// TIA Portal V17 export
// export: Created 2024-09-03T21:54:57.3136222Z, ExportSetting WithDefaults, DisplayName Totally Integrated Automation Portal, DisplayVersion V17 Update 7, DisplayName TIA Portal Openness, DisplayVersion V17 Update 7, DisplayName TIA Portal Version Control Interface, DisplayVersion V17, DisplayName SINAMICS Startdrive Advanced, DisplayVersion V17 SP2, DisplayName SINAMICS Startdrive G110M, G120, G120C, G120D, G120P, G115D, DisplayVersion V17 SP2, DisplayName SINAMICS Startdrive G130, G150, S120, S150, SINAMICS MV, S210, DisplayVersion V17 SP2, DisplayName STEP 7 Professional, DisplayVersion V17 Update 7, DisplayName STEP 7 Safety, DisplayVersion V17 Update 6, DisplayName WinCC Advanced / Unified PC, DisplayVersion V17 Update 7
DATA_BLOCK "AlarmsHandling_DB"   // DB16
VERSION : 0.1
// stored: AutoNumber true, DBAccessibleFromOPCUA true, DBAccessibleFromWebserver true, InstanceOfName AlarmsHandling, InstanceOfType FB
"AlarmsHandling"
   // VAR
   //    IEC_Timer_0_Instance_4 { S7_SetPoint := 'True'} : TON_TIME;
   //    IEC_Timer_0_Instance_5 { S7_SetPoint := 'True'} : TP_TIME;
   //    SetAlarmInstance { S7_SetPoint := 'True'} : Array[0..100] of "SetAlarm_PLC";
   //    AlarmPLCset { S7_SetPoint := 'True'} : Array[0..100] of Program_Alarm;
   // END_VAR
BEGIN
   IEC_Timer_0_Instance_4.PT := T#3S;
   IEC_Timer_0_Instance_4.IN := FALSE;
   IEC_Timer_0_Instance_5.PT := T#0MS;
   IEC_Timer_0_Instance_5.IN := FALSE;
   SetAlarmInstance[0..100].iAlarmCondition := FALSE;
   SetAlarmInstance[0..100].iReset := FALSE;
   SetAlarmInstance[0..14].iTime := T#0MS;
   SetAlarmInstance[15].iTime := T#8S;
   SetAlarmInstance[16..19].iTime := T#5S;
   SetAlarmInstance[20].iTime := T#0MS;
   SetAlarmInstance[21..24].iTime := T#5S;
   SetAlarmInstance[25].iTime := T#0MS;
   SetAlarmInstance[26..28].iTime := T#5S;
   SetAlarmInstance[29..100].iTime := T#0MS;
   SetAlarmInstance[0..100].AlarmToSet := FALSE;
   SetAlarmInstance[0..17].IEC_Timer_0_Instance.PT := T#0MS;
   SetAlarmInstance[18..19].IEC_Timer_0_Instance.PT := T#5S;
   SetAlarmInstance[20..100].IEC_Timer_0_Instance.PT := T#0MS;
   SetAlarmInstance[0..100].IEC_Timer_0_Instance.IN := FALSE;
   SetAlarmInstance[0..100].AlarmToSetWork := FALSE;
END_DATA_BLOCK
